// TIA Portal V17 export
// export: Created 2022-06-27T14:01:33.4642816Z, ExportSetting WithDefaults, DisplayName Totally Integrated Automation Portal, DisplayVersion V17 Update 3, DisplayName TIA Portal Openness, DisplayVersion V17 Update 3, DisplayName TIA Portal Version Control Interface, DisplayVersion V17, DisplayName SINAMICS Startdrive Advanced, DisplayVersion V17 Update1, DisplayName SINAMICS Startdrive G110M, G120, G120C, G120D, G120P, G115D, DisplayVersion V17 Update1, DisplayName SINAMICS Startdrive G130, G150, S120, S150, SINAMICS MV, S210, DisplayVersion V17 Update1, DisplayName STEP 7 Professional, DisplayVersion V17 Update 3, DisplayName STEP 7 Safety, DisplayVersion V17, DisplayName WinCC UA Professional, DisplayVersion V17 Update 3
VAR_GLOBAL   // PLC tag table "Default tag table"
   "EnergyMeterUnkown(1)" AT %IW190 : Int;
   "EnergyMeterUnkown(2)" AT %IW192 : Int;
   "EnergyMeterUnkown(3)" AT %IW194 : Int;
   "EnergyMeterUnkown(4)" AT %QW4 : Int;
   "EnergyMeterUnkown(5)" AT %QW6 : Int;
   "EnergyMeterUnkown(6)" AT %QW8 : Int;
   "EnergyMeterUnkown(7)" AT %QW10 : Int;
   "EnergyMeterUnkown(8)" AT %QW12 : Int;
   "EnergyMeterUnkown(9)" AT %QW14 : Int;
   Clock_Byte AT %MB0 : Byte;
   Clock_10Hz AT %M0.0 : Bool;
   Clock_5Hz AT %M0.1 : Bool;
   "Clock_2.5Hz" AT %M0.2 : Bool;
   Clock_2Hz AT %M0.3 : Bool;
   "Clock_1.25Hz" AT %M0.4 : Bool;
   Clock_1Hz AT %M0.5 : Bool;
   "Clock_0.625Hz" AT %M0.6 : Bool;
   "Clock_0.5Hz" AT %M0.7 : Bool;
END_VAR
